// TIA Portal V20 export
DATA_BLOCK "DB_WorkingModes"   // DB100
// stored: InstanceOfName FB_WorkingModes, InstanceOfType FB
"FB_WorkingModes"
   // VAR_INPUT
   //    iChangeModeEnable : Bool;
   // END_VAR
   // VAR_IN_OUT
   //    ioEmptyingReq : Bool;
   //    ioAutoReq : Bool;
   //    ioSemiAutoReq : Bool;
   //    ioManuReq : Bool;
   // END_VAR
   // VAR
   //    sRT_Filling : R_TRIG;
   //    sRT_Normal { S7_SetPoint := 'True'} : R_TRIG;
   //    sRT_Emptying { S7_SetPoint := 'True'} : R_TRIG;
   //    sFT_Emptying { S7_SetPoint := 'True'} : F_TRIG;
   //    sRT_Auto { S7_SetPoint := 'True'} : R_TRIG;
   //    sRT_SemiAuto { S7_SetPoint := 'True'} : R_TRIG;
   //    sRT_Manu { S7_SetPoint := 'True'} : R_TRIG;
   //    sFilling { S7_SetPoint := 'True'} : Bool;
   //    sNormal : Bool;
   //    sEmptying : Bool;
   //    sAuto : Bool;
   //    sSemiAuto : Bool;
   //    sManu : Bool;
   //    sOnePiece : Bool;
   //    sDryRun : Bool;
   // END_VAR
BEGIN
END_DATA_BLOCK
